FUNCTION_BLOCK FB_CAN_LV
VAR_INPUT
END_VAR
VAR_OUTPUT
END_VAR
VAR
	stBattery1 AT %I* : ST_FMB_BatteryData;
END_VAR

END_FUNCTION_BLOCK

(* stored: Version 1.1.0.1
   POU FB_CAN_LV: Id {3a661af8-15ae-4798-b6ff-82d9d1802389}, SpecialFunc None *)
